{attribute 'estimated-stack-usage' := '4096'}
FUNCTION INTERNAL F_WriteRepeatedField : HRESULT
VAR_IN_OUT
    stCtx  : ST_WriteContext;
END_VAR
VAR_INPUT CONSTANT
	ipRepeatedField	: I_RepeatedField;
END_VAR

VAR
    nPackedDataSize : UDINT;
    i               : UDINT;
    hr              : HRESULT;
    anyItem         : T_Any;
	nTag			: UDINT;
	nEndTag			: UDINT;
END_VAR

IF ipRepeatedField.ipFieldCodec = 0  THEN
	F_WriteRepeatedField := F_WriteError(stCtx, E_WriterErrorCode.InternalError);
    RETURN;
END_IF

IF ipRepeatedField.nCapcacity = 0 OR ipRepeatedField.nCount = 0 THEN
	RETURN;
END_IF

nTag := ipRepeatedField.ipFieldCodec.Tag;
nEndTag := ipRepeatedField.ipFieldCodec.EndTag;

IF ipRepeatedField.ipFieldCodec.IsPackedRepeatedField(nTag)  THEN
    // packed: tag, length, and value
    
    hr := F_WriteRawVarint32(stCtx, nTag);
    IF FAILED(hr) THEN
        F_WriteRepeatedField := hr;
        RETURN;
    END_IF
    
    hr := ipRepeatedField.CalculatePackedDataSize( nPackedDataSize=> nPackedDataSize);
	IF FAILED(hr) THEN
        F_WriteRepeatedField := hr;
        RETURN;
    END_IF
    
    hr := F_WriteLength(stCtx, nPackedDataSize);
    IF FAILED(hr) THEN
        F_WriteRepeatedField := hr;
        RETURN;
    END_IF
    
    FOR i := 0 TO ipRepeatedField.nCount - 1 DO
 		anyItem := ipRepeatedField.ElementAtIndex(i);
        hr := ipRepeatedField.ipFieldCodec.ValueWriter(stCtx, anyItem);
        IF FAILED(hr) THEN
            F_WriteRepeatedField := hr;
            RETURN;
        END_IF
    END_FOR
    
ELSE    
   // Not packed: a simple tag/value pair for each value.
    FOR i := 0 TO ipRepeatedField.nCount - 1 DO
		
		// Write Tag
        hr := F_WriteRawVarint32(stCtx, nTag);
        IF FAILED(hr) THEN
            F_WriteRepeatedField := hr;
            RETURN;
        END_IF
        
 		anyItem := ipRepeatedField.ElementAtIndex(i);
        hr := ipRepeatedField.ipFieldCodec.ValueWriter(stCtx, anyItem);
        IF FAILED(hr) THEN
            F_WriteRepeatedField := hr;
            RETURN;
        END_IF
		
		IF nEndTag <> 0 THEN
			hr := F_WriteRawVarint32(stCtx, nEndTag);
			IF FAILED(hr) THEN
				F_WriteRepeatedField := hr;
				RETURN;
			END_IF			
		END_IF
    END_FOR
END_IF

END_FUNCTION

(* stored: Version 1.1.0.1
   POU F_WriteRepeatedField: Id {663074d2-db41-414f-a82e-bae95a3038e4}, SpecialFunc None *)
